TYPE StationCounters :
STRUCT
	Idle_Counter : UDINT := 0;
	Process_Counter : UDINT := 0;
	Waiting_Counter : UDINT := 0;
END_STRUCT
END_TYPE

(* stored: Version 1.1.0.1, ProductVersion 3.1.0.36
   DUT StationCounters: Id {20519793-8075-495b-bf2e-f4c3702a951e} *)
